(* IEC 61131-3 sources: mastertool-rankine-bridge/tests/indexer/fixtures/sample_export/objects/application_gvl_0__GvlMotoresSintetica, 1 file *)

(* ---- declaration.st ---- *)
{attribute 'qualified_only'}
VAR_GLOBAL
END_VAR
VAR_GLOBAL RETAIN
    MT01: Motor;
    MT02: Motor;
END_VAR
VAR_GLOBAL
    MT03: Motor;
    MT04_ComEndereco AT %QX54.0 : BOOL := TRUE;
END_VAR
